Fanuc KAREL source: ka00122.KL

PROGRAM KA00122
%NOLOCKGROUP
VAR
SRC : ARRAY[2] OF BYTE
DST:REAL
BEGIN
SRC[1]=2
DST=(SRC[1])
END KA00122
